(* Logix 5000 project; controller projeto_base Emulate 5570 rev 19.11; software revision 19.01 *)

TASK MainTask (continuous, watchdog 500 ms) : MainProgram

MODULES
   Local : Emulate 5570 (ICP 2, rev 19.11)
END_MODULES

VAR_GLOBAL   (* controller tags *)
   DESLIGA : BOOL;
   LIGA : BOOL;
   MOTOR1 : BOOL;
END_VAR

PROGRAM MainProgram   (* main routine MainRoutine *)

ROUTINE MainRoutine   (* ladder *)
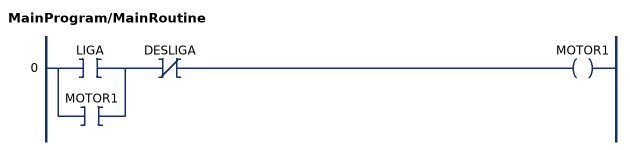
   0: [XIC(LIGA) ,XIC(MOTOR1) ]XIO(DESLIGA)OTE(MOTOR1);
END_ROUTINE
END_PROGRAM
